# B&R Automation Studio project OTTO_Introduction
Automation Studio 4.7.2.98

## Configuration Attachment_ModbusGPIO

### Task classes (Cpu.sw)
```
Cyclic#1 (cycle 10000 us, tolerance 10000 us):
  Handshake <- Handshake.prg
Cyclic#4 (cycle 100000 us, tolerance 100000 us):
  Modbus <- Modbus.prg
Binaries: udbdef, FWRules, TCData, iomap, ashwac, Role, sysconf, arconfig, asfw, User, ashwd
Libraries: standard, runtime, AsOpcUac, astime, asieccon
```

### Hardware
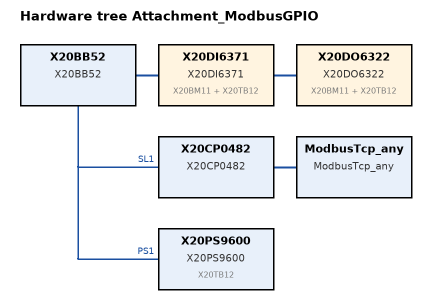
```
ModbusTcp_any : ModbusTcp_any v1.0.6.0  [ETH1 -> X20CP0482.IF2 [Cable Type=PowerlinkCable, Length=10, Version=1.0.0.2]]
  IpAddress = 10.252.252.1  // OTTO's IP 
X20BB52 : X20BB52 v1.1.1.0
X20BM11 : X20BM11 v1.0.0.1  [X2X1 -> X20BB52.IF6]
X20BM11a : X20BM11 v1.0.0.1  [X2X1 -> X20BM11.X2X2]
X20CP0482 : X20CP0482 v1.4.2.0  [SL -> X20BB52.SL1]
  Connector IF2:
    ActivateDevice = 1
    Mode = Manual
    InternetAddress = 10.252.252.10  // B&R PLC's IP
    SubnetMask = 255.255.255.0
    ActivateModbus = 1
    NumSlaves = -1
    NumAllBlocks = -1
    MemSizeIn = -1
    MemSizeOut = -1
    ModbusSlaveGrey = 1
    ModbusSlaveConfig_1
    CoilChannelGroup1_1
    CoilChannelID1_1 = Safe_To_Move
    CoilChannelAddress1_1 = 4000
    HoldingRegisterChannelGroup1_1
    HoldingRegisterChannelID1_1 = attachment_type
    HoldingRegisterChannelAddress1_1 = 4004
    HoldingRegisterChannelType1_1 = UINT
    ModbusMaster = 0
  ConfigurationID = OTTO_Config1
  TimerDeviceType = SWIOTIMER
  Cyclic1Duration = 10000
  Cyclic1Tolerance = 10000
  Cyclic2Duration = 20000
  Cyclic2Tolerance = 20000
  Cyclic3Duration = 50000
  Cyclic3Tolerance = 50000
  Cyclic4Duration = 100000
  Cyclic4Tolerance = 100000
  Cyclic5Duration = 200000
  Cyclic5Tolerance = 200000
  Cyclic6Duration = 500000
  Cyclic6Tolerance = 500000
  Cyclic7Duration = 1000000
  Cyclic7Tolerance = 1000000
  Cyclic8Duration = 10000
  Cyclic8Tolerance = 30000000
X20DI6371 : X20DI6371 v1.0.2.0  [SS1 -> X20TB12a.SS; SL -> X20BM11.SL1]
X20DO6322 : X20DO6322 v1.0.4.0  [SS1 -> X20TB12b.SS; SL -> X20BM11a.SL1]
X20PS9600 : X20PS9600 v1.2.0.0  [PS -> X20BB52.PS1; SS1 -> X20TB12.SS]
X20TB12 : X20TB12 v1.0.0.0
X20TB12a : X20TB12 v1.0.0.0
X20TB12b : X20TB12 v1.0.0.0
```

## Configuration Config1

### Task classes (Cpu.sw)
```
Cyclic#1 (cycle 10000 us, tolerance 10000 us):
  Handshake <- Libraries.Handshake.prg
Cyclic#4 (cycle 100000 us, tolerance 100000 us):
  Modbus <- Modbus.prg
Binaries: udbdef, FWRules, TCData, iomap, ashwac, Role, sysconf, arconfig, asfw, User, ashwd
Libraries: standard, astime, asieccon, runtime
```

### Hardware
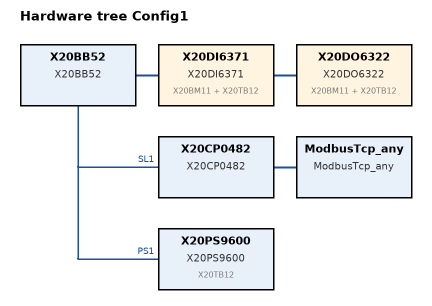
```
ModbusTcp_any : ModbusTcp_any v1.0.6.0  [ETH1 -> X20CP0482.IF2 [Cable Type=PowerlinkCable, Length=10, Version=1.0.0.2]]
  IpAddress = 10.252.252.1  // OTTO's IP
X20BB52 : X20BB52 v1.1.1.0
X20BM11 : X20BM11 v1.0.0.1  [X2X1 -> X20BB52.IF6]
X20BM11a : X20BM11 v1.0.0.1  [X2X1 -> X20BM11.X2X2]
X20CP0482 : X20CP0482 v1.4.2.0  [SL -> X20BB52.SL1]
  Connector IF2:
    ActivateDevice = 1
    Mode = Manual  //  10.252.252.10 (port 502).
    InternetAddress = 10.252.252.10  // PLC's IP
    SubnetMask = 255.255.255.0
    ActivateModbus = 1
    NumSlaves = -1
    NumAllBlocks = -1
    MemSizeIn = -1
    MemSizeOut = -1
    ModbusSlaveGrey = 1
    ModbusSlaveConfig_1
    CoilChannelGroup1_1
    CoilChannelID1_1 = Safe_To_Move
    CoilChannelAddress1_1 = 4000
    HoldingRegisterChannelGroup1_1
    HoldingRegisterChannelID1_1 = attachment_type
    HoldingRegisterChannelAddress1_1 = 4004  // A Holding Register Start Offset of 3999 is required to shift the address range to that which the OTTO SDV expects.
    HoldingRegisterChannelType1_1 = UINT
    ModbusMaster = 0
    SlaveDiagnostics = 2
    IpAddressLow = 10.252.252.1
  Connector IF3:
    Operation = EthOnly
    EthernetMode = DHCPServer
    InternetAddress = 169.254.39.254
    SubnetMask = 255.255.255.0
    ActivateIna = 1
    ActivateANSL = 1
  ConfigurationID = OTTO_Config1
  TimerDeviceType = SWIOTIMER
  Cyclic1Duration = 10000
  Cyclic1Tolerance = 10000
  Cyclic2Duration = 20000
  Cyclic2Tolerance = 20000
  Cyclic3Duration = 50000
  Cyclic3Tolerance = 50000
  Cyclic4Duration = 100000
  Cyclic4Tolerance = 100000
  Cyclic5Duration = 200000
  Cyclic5Tolerance = 200000
  Cyclic6Duration = 500000
  Cyclic6Tolerance = 500000
  Cyclic7Duration = 1000000
  Cyclic7Tolerance = 1000000
  Cyclic8Duration = 10000
  Cyclic8Tolerance = 30000000
X20DI6371 : X20DI6371 v1.0.2.0  [SS1 -> X20TB12a.SS; SL -> X20BM11.SL1]
X20DO6322 : X20DO6322 v1.0.4.0  [SS1 -> X20TB12b.SS; SL -> X20BM11a.SL1]
X20PS9600 : X20PS9600 v1.2.0.0  [PS -> X20BB52.PS1; SS1 -> X20TB12.SS]
X20TB12 : X20TB12 v1.0.0.0
X20TB12a : X20TB12 v1.0.0.0
X20TB12b : X20TB12 v1.0.0.0
```

### IoMap.iom - X20CP0482/IoMap.iom
```iecst
VAR_CONFIG
	::Handshake:io.handshake.PA_ENABLE AT %IX."X20DI6371".DigitalInput01 INVERSE;
	::Handshake:io.handshake.ROBOT_ENABLE AT %QX."X20DO6322".DigitalOutput01;
	::Handshake:io.handshake.PA_FAULT_STATUS AT %QX."X20DO6322".DigitalOutput02;
	::Handshake:io.LED AT %QX."X20DO6322".DigitalOutput06;
	::Modbus:modbus.Attachment_Type AT %IW."X20CP0482".IF2.attachment_type;
	::Modbus:modbus.Attachment_Type AT %QW."ModbusTcp_any".attachment_type;
	::Modbus:modbus.Safe_to_Move AT %IX."ModbusTcp_any".safe_to_move;
	::Modbus:modbus.Safe_to_Move AT %IX."X20CP0482".IF2.Safe_To_Move;
END_VAR
```

## Configuration ModbusForIgnition

CPU X20CP0482, AutomationRuntime A4.73, Build 4.1.2, Vc V4.72.0

### Hardware
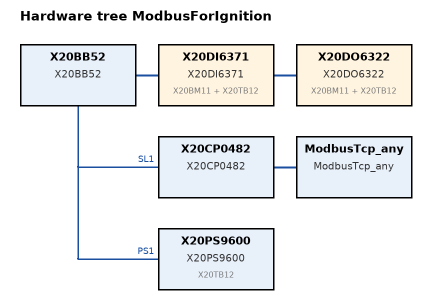
```
ModbusTcp_any : ModbusTcp_any v1.0.6.0  [ETH1 -> X20CP0482.IF2 [Cable Type=PowerlinkCable, Length=10, Version=1.0.0.2]]
  IpAddress = 192.168.1.230  // Ignition's Gateway IP
  Cb_1
  Cb_1_FunCode = 6
  Cb_1_C_1
  Cb_1_C_1_Name = mission_create_0
  Cb_1_C_1_Datatype = 6
  Cb_1_C_1_Dir = 1
X20BB52 : X20BB52 v1.1.1.0
X20BM11 : X20BM11 v1.0.0.1  [X2X1 -> X20BB52.IF6]
X20BM11a : X20BM11 v1.0.0.1  [X2X1 -> X20BM11.X2X2]
X20CP0482 : X20CP0482 v1.4.2.0  [SL -> X20BB52.SL1]
  Connector IF2:
    ActivateDevice = 1
    Mode = Manual
    InternetAddress = 192.168.1.230  // B&R PLC's IP
    SubnetMask = 255.255.255.0
    ActivateModbus = 1
    NumSlaves = -1
    NumAllBlocks = -1
    MemSizeIn = -1
    MemSizeOut = -1
    ModbusSlaveGrey = 1
    ModbusSlaveConfig_1
    HoldingRegisterChannelGroup1_1
    HoldingRegisterChannelID1_1 = Mission_create_0
    HoldingRegisterChannelAddress1_1 = 0
    HoldingRegisterChannelType1_1 = UINT
  ConfigurationID = OTTO_Config1
  TimerDeviceType = SWIOTIMER
  Cyclic1Duration = 10000
  Cyclic1Tolerance = 10000
  Cyclic2Duration = 20000
  Cyclic2Tolerance = 20000
  Cyclic3Duration = 50000
  Cyclic3Tolerance = 50000
  Cyclic4Duration = 100000
  Cyclic4Tolerance = 100000
  Cyclic5Duration = 200000
  Cyclic5Tolerance = 200000
  Cyclic6Duration = 500000
  Cyclic6Tolerance = 500000
  Cyclic7Duration = 1000000
  Cyclic7Tolerance = 1000000
  Cyclic8Duration = 10000
  Cyclic8Tolerance = 30000000
X20DI6371 : X20DI6371 v1.0.2.0  [SS1 -> X20TB12a.SS; SL -> X20BM11.SL1]
X20DO6322 : X20DO6322 v1.0.4.0  [SS1 -> X20TB12b.SS; SL -> X20BM11a.SL1]
X20PS9600 : X20PS9600 v1.2.0.0  [PS -> X20BB52.PS1; SS1 -> X20TB12.SS]
X20TB12 : X20TB12 v1.0.0.0
X20TB12a : X20TB12 v1.0.0.0
X20TB12b : X20TB12 v1.0.0.0
```

### IoMap.iom - X20CP0482/IoMap.iom
```iecst
VAR_CONFIG
	::Handshake:io.handshake.ROBOT_ENABLE AT %QX."X20DO6322".DigitalOutput01;
	::Handshake:io.handshake.PA_FAULT_STATUS AT %QX."X20DO6322".DigitalOutput02;
	::Handshake:io.LED AT %QX."X20DO6322".DigitalOutput06;
	::Handshake:io.handshake.PA_ENABLE AT %IX."X20DI6371".DigitalInput01 INVERSE;
	::Modbus:modbus.Mission_create_0 AT %IW."X20CP0482".IF2.Mission_create_0;
	::Modbus:modbus.Create_mission_1 AT %IW."X20CP0482".IF2.Mission_create_1;
	::Modbus:modbus.Attachment_Type AT %QW."ModbusTcp_any".attachment_type;
	::Modbus:modbus.Safe_to_Move AT %IX."ModbusTcp_any".safe_to_move;
	::Modbus:modbus.Mission_create_0 AT %QW."ModbusTcp_any".mission_create_0;
	::Modbus:modbus.Create_mission_1 AT %IO."X20CP0482".IF2.Mission_create_1;
	::Modbus:io.Mission_startButton AT %IX."X20DI6371".DigitalInput02;
END_VAR
```

## Configuration ModbusGPIO

### Task classes (Cpu.sw)
```
Cyclic#1 (cycle 10000 us, tolerance 10000 us):
  Handshake <- Handshake.prg
Cyclic#4 (cycle 100000 us, tolerance 100000 us):
  Modbus <- Modbus.prg
  Client <- OPC_UA.Client.prg [disabled]
Binaries: udbdef, FWRules, TCData, iomap, ashwac, Role, sysconf, arconfig, asfw, User, ashwd
Libraries: standard, runtime, AsOpcUac, astime, asieccon
```

### Hardware
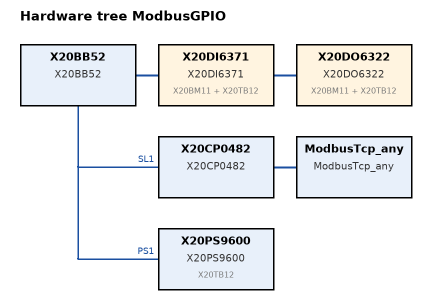
```
ModbusTcp_any : ModbusTcp_any v1.0.6.0  [ETH1 -> X20CP0482.IF2 [Cable Type=PowerlinkCable, Length=10, Version=1.0.0.2]]
  IpAddress = 10.252.252.1  // OTTO's IP
X20BB52 : X20BB52 v1.1.1.0
X20BM11 : X20BM11 v1.0.0.1  [X2X1 -> X20BB52.IF6]
X20BM11a : X20BM11 v1.0.0.1  [X2X1 -> X20BM11.X2X2]
X20CP0482 : X20CP0482 v1.4.2.0  [SL -> X20BB52.SL1]
  Connector IF2:
    ActivateDevice = 1
    Mode = Manual
    InternetAddress = 10.252.252.10
    SubnetMask = 255.255.255.0
    ActivateModbus = 1
    NumSlaves = -1
    NumAllBlocks = -1
    MemSizeIn = -1
    MemSizeOut = -1
    ModbusSlaveGrey = 1
    ModbusSlaveConfig_1
    CoilChannelGroup1_1
    CoilChannelID1_1 = Safe_To_Move
    CoilChannelAddress1_1 = 4000
    HoldingRegisterChannelGroup1_1
    HoldingRegisterChannelID1_1 = attachment_type
    HoldingRegisterChannelAddress1_1 = 4004
    HoldingRegisterChannelType1_1 = UINT
    ModbusMaster = 0
  ConfigurationID = OTTO_Config1
  TimerDeviceType = SWIOTIMER
  Cyclic1Duration = 10000
  Cyclic1Tolerance = 10000
  Cyclic2Duration = 20000
  Cyclic2Tolerance = 20000
  Cyclic3Duration = 50000
  Cyclic3Tolerance = 50000
  Cyclic4Duration = 100000
  Cyclic4Tolerance = 100000
  Cyclic5Duration = 200000
  Cyclic5Tolerance = 200000
  Cyclic6Duration = 500000
  Cyclic6Tolerance = 500000
  Cyclic7Duration = 1000000
  Cyclic7Tolerance = 1000000
  Cyclic8Duration = 10000
  Cyclic8Tolerance = 30000000
X20DI6371 : X20DI6371 v1.0.2.0  [SS1 -> X20TB12a.SS; SL -> X20BM11.SL1]
X20DO6322 : X20DO6322 v1.0.4.0  [SS1 -> X20TB12b.SS; SL -> X20BM11a.SL1]
X20PS9600 : X20PS9600 v1.2.0.0  [PS -> X20BB52.PS1; SS1 -> X20TB12.SS]
X20TB12 : X20TB12 v1.0.0.0
X20TB12a : X20TB12 v1.0.0.0
X20TB12b : X20TB12 v1.0.0.0
```

### IoMap.iom - X20CP0482/IoMap.iom
```iecst
VAR_CONFIG
	::Modbus:modbus.Attachment_Type AT %QW."ModbusTcp_any".attachment_type;
	::Modbus:modbus.Safe_to_Move AT %IX."ModbusTcp_any".safe_to_move;
	::Handshake:io.handshake.ROBOT_ENABLE AT %QX."X20DO6322".DigitalOutput01;
	::Handshake:io.handshake.PA_FAULT_STATUS AT %QX."X20DO6322".DigitalOutput02;
	::Handshake:io.LED AT %QX."X20DO6322".DigitalOutput06;
	::Handshake:io.handshake.PA_ENABLE AT %IX."X20DI6371".DigitalInput01 INVERSE;
END_VAR
```

## Configuration OPCforIgnition

CPU X20CP0482, AutomationRuntime A4.73, Build 4.1.2, Vc V4.72.0

### Task classes (Cpu.sw)
```
Cyclic#4 (cycle 100000 us, tolerance 100000 us):
  Server <- OPC_UA.Server.prg
Binaries: udbdef, FWRules, TCData, sysconf, Role, User, iomap, ashwd, asfw, arconfig, ashwac, Config
Libraries: AsOpcUas, runtime, AsOpcUac, astime, asieccon
```

### Hardware
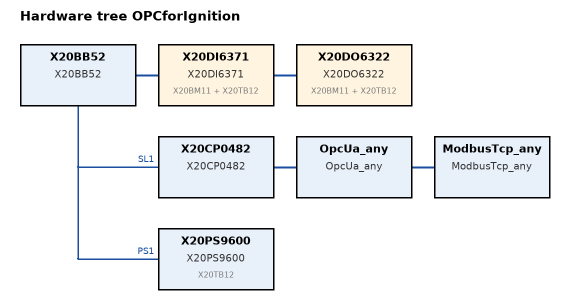
```
ModbusTcp_any : ModbusTcp_any v1.0.6.0  [ETH1 -> OpcUa_any.ETH2 [Cable Type=PowerlinkCable, Length=10, Version=1.0.0.2]]
  IpAddress = 192.168.1.7
OpcUa_any : OpcUa_any v1.0.0.1  [ETH1 -> X20CP0482.IF2 [Cable Type=PowerlinkCable, Length=10, Version=1.0.0.2]; ETH2 -> ModbusTcp_any.ETH1 [Cable Type=PowerlinkCable, Length=10, Version=1.0.0.2]]
  ServerDiagnostics = on
  ServerEndpointUrl = opc.tcp://192.168.1.230:4841
  OpcUa_Security_SoftwareCertificates = SSLConfiguration
X20BB52 : X20BB52 v1.1.1.0
X20BM11 : X20BM11 v1.0.0.1  [X2X1 -> X20BB52.IF6]
X20BM11a : X20BM11 v1.0.0.1  [X2X1 -> X20BM11.X2X2]
X20CP0482 : X20CP0482 v1.4.2.0  [SL -> X20BB52.SL1]
  Connector IF2:
    ActivateDevice = 1
    Mode = Manual
    InternetAddress = 192.168.1.230
    SubnetMask = 255.255.0.0
    ActivateModbus = 1
    NumSlaves = -1
    NumAllBlocks = -1
    MemSizeIn = -1
    MemSizeOut = -1
    ModbusSlaveGrey = 1
    ModbusMaster = 0
  Connector IF3:
    Operation = EthOnly
    EthernetMode = DHCPServer
    InternetAddress = 169.254.39.254
    SubnetMask = 255.255.255.0
    ActivateIna = 1
    ActivateANSL = 1
  ConfigurationID = OPC_server
  ApplicationStorageType = NORMAL
  SimulationModeOpcUa = off
  Connections = 5
  TimerDeviceType = SWIOTIMER
  Cyclic1Duration = 10000
  Cyclic1Tolerance = 10000
  Cyclic2Duration = 20000
  Cyclic2Tolerance = 20000
  Cyclic3Duration = 50000
  Cyclic3Tolerance = 50000
  Cyclic4Duration = 100000
  Cyclic4Tolerance = 100000
  Cyclic5Duration = 200000
  Cyclic5Tolerance = 200000
  Cyclic6Duration = 500000
  Cyclic6Tolerance = 500000
  Cyclic7Duration = 1000000
  Cyclic7Tolerance = 1000000
  Cyclic8Duration = 10000
  Cyclic8Tolerance = 30000000
  TimeZone = 150
  ActivateFtpServer = 0
  ActivateTftpServer = 0
  ActivateSdm = 0
  ActivateOpcUa = 1
  OpcUaPort = 4841
  OpcUa_AuthenticationSecurityPolicy_EnableNone = 1
  OpcUa_AuthenticationSecurityPolicy_EnableBasic128Rsa15 = 1
  OpcUa_Security_AdminRole = 
  OpcUa_Security_SoftwareCertificates = SSLConfiguration
  OpcUaInformationModels_PV_Version = 2
X20DI6371 : X20DI6371 v1.0.2.0  [SS1 -> X20TB12a.SS; SL -> X20BM11.SL1]
X20DO6322 : X20DO6322 v1.0.4.0  [SS1 -> X20TB12b.SS; SL -> X20BM11a.SL1]
X20PS9600 : X20PS9600 v1.2.0.0  [PS -> X20BB52.PS1; SS1 -> X20TB12.SS]
X20TB12 : X20TB12 v1.0.0.0
X20TB12a : X20TB12 v1.0.0.0
X20TB12b : X20TB12 v1.0.0.0
```

### MyRequest.csr - X20CP0482/AccessAndSecurity/CertificateStore/CertificateSigningRequests/MyRequest.csr
```
-----BEGIN CERTIFICATE REQUEST-----
MIICLzCCAZigAwIBAgIQTWihe8Pw/55FXlhwKpR/tzANBgkqhkiG9w0BAQ0FADAy
MSMwIQYJKoZIhvcNAQkBFhRtc3ZAbm9yZC1tb2R1bGVzLmNvbTELMAkGA1UEBhMC
REswHhcNMjAxMjExMDAwMDAwWhcNMjIxMjExMTExOTE1WjAyMSMwIQYJKoZIhvcN
AQkBFhRtc3ZAbm9yZC1tb2R1bGVzLmNvbTELMAkGA1UEBhMCREswgZ8wDQYJKoZI
hvcNAQEBBQADgY0AMIGJAoGBAMFVN/waFnn+caNAUlnqtAMGp95CF4tO/1O8RCyg
R+wst6WgXAvvbWiMTFYLYX3GFNvWchXQD3AnGu1ZzDIxFtkzAUaoqjS2oBUWRJfz
fzPR+NAyWgH5cEle4bkRBVIqx6R+Mo65xcZ/BCmwksckK3ZJ0df/7QwVkmKnq9Lx
D6GxAgMBAAGjRjBEMBMGA1UdJQQMMAoGCCsGAQUFBwMCMB0GA1UdDgQWBBSUJB7W
xwcX9dY056zGYZpAr5mGZjAOBgNVHQ8BAf8EBAMCB4AwDQYJKoZIhvcNAQENBQAD
gYEAkkWKDe7BKONzrQf/evalJhEUBZORkfq2XfFGkE6Ou+4slfOdGe7QRNwbcGWs
3nnCZvp03BBTBDExd64h21MZPazkbTAOT+oi6ZF3cnOj5vecstR087q+LTxlPw16
o4f8Z5osTaDu+idu83rBLXO2r1uPIJMJ7jJDb+qEKnurNks=
-----END CERTIFICATE REQUEST-----
```

### OpcUa.uanodeset - X20CP0482/Connectivity/OpcUA/OpcUa.uanodeset
```
UANodeSet:
  NamespaceUris:
    Uri = http://inductiveautomation.com/products/ignitionopc/
  Aliases:
    Alias = i=1 (Alias=Boolean)
    Alias = i=2 (Alias=SByte)
    Alias = i=3 (Alias=Byte)
    Alias = i=4 (Alias=Int16)
    Alias = i=5 (Alias=UInt16)
    Alias = i=6 (Alias=Int32)
    Alias = i=7 (Alias=UInt32)
    Alias = i=12 (Alias=String)
```

### IoMap.iom - X20CP0482/IoMap.iom
```iecst
VAR_CONFIG
	::Server:Test_Variable1 AT %QX."X20DO6322".DigitalOutput03;
	::Server:Test_Variable2 AT %QX."X20DO6322".DigitalOutput04;
	::Server:Test_Variable3 AT %QX."X20DO6322".DigitalOutput05;
END_VAR
```

### OpcArMap.opcc - X20CP0482/OpcArMap.opcc
```
Map:
  Tag Test_Variable2 (Scope=OPC_UA)
    PV Test_Variable2 (Task=Server, DataType=boolean, IsVector=False, BitNumber=none)
  Tag Test_Variable1 (Scope=OPC_UA)
    PV Test_Variable1 (Task=Server, DataType=boolean, IsVector=False, BitNumber=none)
```

## Logical view

Binary libraries used (declarations not repeated): operator, runtime, standard, astime, AsIecCon, AsOpcUac, AsOpcUas

### Package Logical/Libraries - Global libraries

### Program Logical/Libraries/Handshake

#### Types.typ
```iecst
TYPE
	GPIO_Hanshake_type : 	STRUCT
		ROBOT_ENABLE : BOOL;
		PA_FAULT_STATUS : BOOL;
		PA_ENABLE : BOOL;
	END_STRUCT;
	io_type : 	STRUCT
		handshake : GPIO_Hanshake_type;
		LED : BOOL;
	END_STRUCT;
END_TYPE
```

#### Variables.var
```iecst
VAR
	io : io_type;
	timer : TON;
END_VAR
```

#### handshake.st
```iecst
PROGRAM _INIT
	(* Insert code here *)
	io.handshake.PA_FAULT_STATUS := TRUE; //No error in the beginning
	io.handshake.ROBOT_ENABLE := TRUE; //Attachnment indicates OTTO has control

	timer.PT := T#1s;

END_PROGRAM

PROGRAM _CYCLIC

	//OTTO GIVES CONTROL TO ATTACHMENT
	IF io.handshake.PA_ENABLE THEN
		io.handshake.ROBOT_ENABLE := FALSE;
		io.LED := TRUE;
		timer.IN := TRUE;
	END_IF;

	//ATTACHMENT GIVES CONTROL BACK TO OTTO
		IF timer.Q THEN
			timer.IN := FALSE;
			io.handshake.ROBOT_ENABLE := TRUE;
			io.LED := FALSE;
		END_IF

	timer();
END_PROGRAM
```

### Program Logical/Modbus (IEC)

#### modbus.st - Cyclic code
```iecst
//Used for Modbus communication with Ignition. Variables and code is used to initialize the mission in fleet
PROGRAM _INIT

END_PROGRAM

PROGRAM _CYCLIC
(* This snippet is not necessary for prototyping and I am not sure how B&R handles overflow, in either case, overflow protection is a good practice!
	IF modbus.Create_mission_0 := 4294967295 THEN// maximum size of UINT (OVERFLOW PROTECTION)
		modbus.Create_mission_0 := 0;
	END_IF
	IF modbus.Create_mission_1 := 4294967295 THEN// maximum size of UINT (OVERFLOW PROTECTION)
		modbus.Create_mission_1 := 0;
	END_IF *)
	IF EDGEPOS (io.Mission_startButton) THEN
		counter := counter + 1;
	END_IF
	modbus.Mission_create_0 := counter  ;

END_PROGRAM
```

#### Types.typ - Local data types
```iecst
TYPE
	io_type : 	STRUCT
		Mission_startButton : BOOL;
	END_STRUCT;
	modbus_type : 	STRUCT
		Attachment_Type : UINT := 10; (*Value uniquely identifying the type of attachment. Unsigned int 16:: 76 LIFT / 67 CONVEYOR*)
		HoldReg : UDINT;
		Safe_to_Move : BOOL;
		Mission_create_0 : UINT;
	END_STRUCT;
END_TYPE
```

#### Variables.var - Local variables
```iecst
VAR
	counter : UINT;
	io : io_type;
	modbus : modbus_type;
END_VAR
```

- Program Logical/Handshake (IEC) (no source held here)

### Program Logical/OPC_UA/Server (IEC)

#### Cyclic.ab - Cyclic code
```automation-basic
PROGRAM _CYCLIC
	//just to check for variables at the moment

END_PROGRAM
```

#### Variables.var - Local variables
```iecst
VAR
	Test_Variable1 : BOOL;
	Test_Variable2 : BOOL;
	Test_Variable3 : BOOL;
END_VAR
```

- OpcTag.opct (not shown)

### Program Logical/OPC_UA/Client (IEC)

#### Types.typ - Local data types
```iecst
TYPE
	opc_steps :
		(
		Retain,
		Connect,
		ConnectionGetStatus,
		GetNamespaceIndex,
		NodeGetHandle,
		NodeGetHandleList,
		SubscriptionCreate,
		MonitoredItemAdd,
		MonitoredItemAddList,
		MonitoredItemOperateList,
		MonitoredItemRemoveList,
		SubscriptionDelete,
		WriteList,
		ReadList,
		NodeReleaseHandle,
		NodeReleaseHandleList,
		ErrorHandling,
		Disconnect
		);
	Structure_type : 	STRUCT
		description : STRING[80];
	END_STRUCT;
END_TYPE
```

Listed in the project but not available here: Logical/Global.typ, Logical/Global.var, Logical/Handshake/handshake.st, Logical/Handshake/Types.typ, Logical/Handshake/Variables.var, Logical/OPC_UA/Variables.var, Logical/OPC_UA/Types.typ, Logical/OPC_UA/Server/Types.typ, Logical/OPC_UA/Client/client_ignition.st, Logical/OPC_UA/Client/Variables.var
